{attribute addProperty BoxType "EL3356-0000-0017"}
{attribute addProperty Id "RMB_StatusAT %I*RMB_Status_25CC6AB61620RMB_Value_INT32AT %I*RMB_Value_INT_1F5759573240RMB_ControlAT %Q*RMB_Control_F68E0F331620WcStateAT %I*WcState_98A4DF7520.250InfoDataAT %I*InfoData_BC63D37F80100"}
{attribute addProperty CRC "1106297898"}
{attribute addProperty SizeInBites "146"}
{attribute addProperty SizeInBytes "18.25"}
TYPE EL3356_16C4FA1F :
STRUCT
	{attribute addProperty Name "RMB_Status"}
	RMB_Status : RMB_Status_25CC6AB6;
	{attribute addProperty Name "RMB_Value_INT32"}
	RMB_Value_INT32 : RMB_Value_INT_1F575957;
	{attribute addProperty Name "RMB_Control"}
	RMB_Control : RMB_Control_F68E0F33;
	{attribute addProperty Name "WcState"}
	WcState : WcState_98A4DF75;
	{attribute addProperty Name "InfoData"}
	InfoData : InfoData_BC63D37F;
END_STRUCT
END_TYPE

(* stored: Version 1.2.0.0, ProductVersion 3.1.4024.9
   DUT EL3356_16C4FA1F: Id {b002a0c1-ea5c-487b-acf6-4ae49eb04b1f} *)
